FUNCTION AssignOutletToTank : Result
VAR_INPUT
	refTank		: REFERENCE TO ARRAY[1..CST.MAX_TANK] OF Tank;
	refOutlet	: REFERENCE TO ARRAY[1..CST.MAX_TANK] OF Outlet;
END_VAR
VAR
	i			: UDINT;
END_VAR

FOR i := 1 TO CST.MAX_TANK DO
	IF IsErr(refOutlet[i].AssignTank(refTank[i]), eCarry => AssignOutletToTank) THEN
		DebugMsg(0, CONCAT('Failed to assign tank to outlet at index ', UDINT_TO_STRING(i)));
	END_IF	
END_FOR

END_FUNCTION

(* stored: Version 1.1.0.1
   POU AssignOutletToTank: Id {7af64d98-5f84-4e04-8d7c-0657abab6c12}, SpecialFunc None *)
